FUNCTION_BLOCK FB_HumiditySensor_EL3054 IMPLEMENTS I_HumiditySensor
VAR_INPUT
END_VAR
VAR_OUTPUT
END_VAR
VAR
	//Property Real value
	fHumidity : REAL;
	//Raw value
	HumRaw AT %I* : INT;
	//Convertion parameters
	m : REAL := 0.00305185071; //Multiplier for convertion
END_VAR

// Humidity measurement with rotronic HygroFlex 5 
// https://www.rotronic.com/de/catalog/product/view/id/299/s/hygroflex5-hf5-hlk-messumformer/category/12/

PROPERTY Humidity : REAL
GET
fHumidity := m* INT_TO_REAL(HumRaw);
Humidity := THIS^.fHumidity;
END_GET
END_PROPERTY

END_FUNCTION_BLOCK

(* stored: Version 1.1.0.1
   POU FB_HumiditySensor_EL3054: Id {0da4b185-c333-42ce-96bc-7d6db4f7a49c}, SpecialFunc None
   Property Humidity: Id {7ba85027-3b4b-485f-aeed-d09726388122}
   Get Get: Id {53f5695d-8143-4b8a-be2e-4d16fcb201b9} *)
